// TIA Portal V16 export
// export: Created 2022-11-17T15:49:47.8701163Z, ExportSetting WithDefaults, DisplayName Totally Integrated Automation Portal, DisplayVersion V16 Update 6, DisplayName TIA Portal Version Control Interface, DisplayVersion V16 Update 2, DisplayName TIA Portal Openness, DisplayVersion V16 Update 6, DisplayName SINAMICS Startdrive Advanced, DisplayVersion V16 Update 5, DisplayName SINAMICS Startdrive G130, G150, S120, S150, SINAMICS MV, S210, DisplayVersion V16 Update 5, DisplayName SINAMICS Startdrive G110M, G120, G120C, G120D, G120P, G115D, DisplayVersion V16 Update 5, DisplayName STEP 7 Professional, DisplayVersion V16 Update 6, DisplayName STEP 7 Safety, DisplayVersion V16, DisplayName WinCC Advanced, DisplayVersion V16 Update 6
VAR_GLOBAL   // PLC tag table "Default tag table"
   "E0.4" AT %I0.4 : Bool;   // CONTROLLO SALDATORE FILM
   "E0.5" AT %I0.5 : Bool;   // RICHIESTA APERTURA PORTA
   "E0.6" AT %I0.6 : Bool;   // PRESSOSTATO MACCHINA
   "E0.7" AT %I0.7 : Bool;   // ALLARME TERMICO MACCHINA
   "E1.0" AT %I1.0 : Bool;   // EMERGENZA MACCHINA
   "E1.1" AT %I1.1 : Bool;   // BARRIERE IMPEGNATE ENTRATA
   "E1.2" AT %I1.2 : Bool;   // BARRIERE IMPEGNATE USCITA
   "E1.3" AT %I1.3 : Bool;   // RESET MACCHINA
   "E1.4" AT %I1.4 : Bool;   // MARCIA AUTOMATICA MACCHINA
   "E1.5" AT %I1.5 : Bool;   // ARRESTO MACCHINA
   "E2.0" AT %I2.0 : Bool;   // TAVOLA IN FASE
   "E2.1" AT %I2.1 : Bool;   // [spare] COMANDO FRENO MOTORE ROTAZIONE
   "E2.2" AT %I2.2 : Bool;   // CARRELLO BASSO
   "E2.3" AT %I2.3 : Bool;   // CARRELLO ALTO
   "E2.4" AT %I2.4 : Bool;   // TAGLIO INDIETRO
   "E2.5" AT %I2.5 : Bool;   // TAGLIO AVANTI
   "E2.6" AT %I2.6 : Bool;   // CONTRASTO SALDATORE INDIETRO
   "E2.7" AT %I2.7 : Bool;   // CONTRASTO SALDATORE BASSO
   "E3.0" AT %I3.0 : Bool;   // RISERVA
   "E3.1" AT %I3.1 : Bool;   // RISERVA
   "E3.2" AT %I3.2 : Bool;   // LETTURA CENTRAGGIO PALLET TRASPORTO CENTRO MACCHINA
   "E3.3" AT %I3.3 : Bool;   // CONTEGGIO CENTRAGGIO PALLET TRASPORTO CENTRO MACCHINA
   "E3.4" AT %I3.4 : Bool;   // CONTROLLO ROTAZIONE TAVOLA IN ENTRATA E LETTURA LUNGHEZZA PALLET
   "E3.5" AT %I3.5 : Bool;   // CONTROLLO ROTAZIONE TAVOLA IN USCITA E FINE CICLO
   "E3.6" AT %I3.6 : Bool;   // SEGNALE PALLET PRONTO IN ENTRATA
   "E3.7" AT %I3.7 : Bool;   // SEGNALE PRONTO A RICEVERE IN USCITA
   "E4.0" AT %I4.0 : Bool;   // SEGNALE FINE TRASFERIMENTO PALLET IN USCITA
   "E4.1" AT %I4.1 : Bool;   // SEGNALE ESCLUSIONE FASCIATURA
   "E4.2" AT %I4.2 : Bool;   // POSIZIONAMENTO PALLET TRASPORTO POS. 01
   "E4.3" AT %I4.3 : Bool;   // POSIZIONAMENTO PALLET TRASPORTO POS. 02
   "E4.4" AT %I4.4 : Bool;   // POSIZIONAMENTO PALLET TRASPORTO POS. 03
   "E4.5" AT %I4.5 : Bool;   // POSIZIONAMENTO PALLET TRASPORTO POS. 04
   "E4.6" AT %I4.6 : Bool;   // POSIZIONAMENTO PALLET TRASPORTO POS. 05
   "E5.1" AT %I5.1 : Bool;   // POSIZIONAMENTO PALLET TRASPORTO POS. 08
   "E5.3" AT %I5.3 : Bool;   // [B2783] CONTROLLO 2 POSIZIONAMENTO POS. 05
   "E6.0" AT %I6.0 : Bool;   // CARRELLO BASSO (TOP)
   "E6.1" AT %I6.1 : Bool;   // CARRELLO ALTO (TOP)
   "E6.2" AT %I6.2 : Bool;   // LETTURA ALTEZZA PALLET (TOP)
   "E6.3" AT %I6.3 : Bool;   // PINZA CHIUSA BLOCCO FILM (TOP)
   "E6.4" AT %I6.4 : Bool;   // TAGLIO FILM AVANTI (TOP)
   "E6.5" AT %I6.5 : Bool;   // TAGLIO FILM INDIETRO (TOP)
   "E6.6" AT %I6.6 : Bool;   // ROTTURA ESAURIMENTO FILM (TOP)
   "E7.0" AT %I7.0 : Bool;   // CARRELLO INDIETRO (TOP)
   "E7.1" AT %I7.1 : Bool;   // CARRELLO AVANTI POSIZIONE TAGLIO (TOP)
   "E7.3" AT %I7.3 : Bool;   // PINZA CHIUSA TRAINO FILM (TOP)
   "E7.4" AT %I7.4 : Bool;   // SICUREZZA AVANZAMENTO (TOP)
   "E7.5" AT %I7.5 : Bool;   // SICUREZZA DISCESA (TOP) SX
   "E7.6" AT %I7.6 : Bool;   // SICUREZZA DISCESA (TOP) DX
   "E7.7" AT %I7.7 : Bool;   // SICUREZZA CONTROLLO SGANCIO FRENI SAL.-DISC. (TOP)
   HSC2Value AT %ID1004 : DInt;   // Counter value for HSC2
   HSC1Value AT %ID1000 : DInt;
   "E4.7" AT %I4.7 : Bool;   // POSIZIONAMENTO PALLET TRASPORTO POS. 06
   "E5.0" AT %I5.0 : Bool;   // POSIZIONAMENTO PALLET TRASPORTO POS. 07
   "E5.2" AT %I5.2 : Bool;   // [B2782] CONTROLLO 1 POSIZIONAMENTO POS. 05
   "E5.4" AT %I5.4 : Bool;   // SEGNALE PORTA TAGLIAFUOCO APERTA
   "E5.5" AT %I5.5 : Bool;   // SEGNALE CHIUSURA PORTA TAGLIAFUOCO
   "E5.6" AT %I5.6 : Bool;   // SelectorBypass
   "E5.7" AT %I5.7 : Bool;   // Free
   "E6.7" AT %I6.7 : Bool;   // SPARE - NOT USED
   "E7.2" AT %I7.2 : Bool;   // RISERVA
   "A0.0" AT %Q0.0 : Bool;   // APERTURA PORTA
   "A0.1" AT %Q0.1 : Bool;   // EMERGENZA PLC SU PILZ
   "A0.2" AT %Q0.2 : Bool;   // EMERGENZA MACCHINA
   "A0.3" AT %Q0.3 : Bool;   // MARCIA AUTOMATICA MACCHINA
   "A0.4" AT %Q0.4 : Bool;   // SEGNALATORE ACUSTICO MARCIA
   "A0.6" AT %Q0.6 : Bool;   // FRENO MOTORE ROTAZIONE
   "A0.7" AT %Q0.7 : Bool;   // MOTORE ROTAZIONE
   "A1.0" AT %Q1.0 : Bool;   // FASCIA STRETTA
   "A1.1" AT %Q1.1 : Bool;   // CORDA STRETTA
   "A2.0" AT %Q2.0 : Bool;   // PINZA APERTA
   "A2.1" AT %Q2.1 : Bool;   // PINZA CHIUSA
   "A2.2" AT %Q2.2 : Bool;   // TAGLIO AVANTI / INDIETRO
   "A2.3" AT %Q2.3 : Bool;   // SOFFIO ARIA PER CODA FILM
   "A2.4" AT %Q2.4 : Bool;   // TAGLIO FILM
   "A2.5" AT %Q2.5 : Bool;   // SALDATORE FILM
   "A2.6" AT %Q2.6 : Bool;   // CONTRASTO SALDATORE AVANTI
   "A2.7" AT %Q2.7 : Bool;   // CONTRASTO SALDATORE INDIETRO
   "A3.0" AT %Q3.0 : Bool;   // CONTRASTO SALDATORE SALITA/DISCESA
   "A3.1" AT %Q3.1 : Bool;   // RISERVA
   "A3.2" AT %Q3.2 : Bool;   // RISERVA
   "A3.3" AT %Q3.3 : Bool;   // MOTORE TRASPORTO CENTRO MACCHINA
   "A3.4" AT %Q3.4 : Bool;   // SEGNALE PRONTO A RICEVERE IN ENTRATA
   "A3.5" AT %Q3.5 : Bool;   // SEGNALE FINE TRASFERIMENTO PALLET IN ENTRATA
   "A3.6" AT %Q3.6 : Bool;   // SEGNALE PALLET PRONTO IN USCITA
   "A3.7" AT %Q3.7 : Bool;   // SEGNALE PRONTO PER CHIUSURA PORTA TAGLIAFUOCO
   "A4.0" AT %Q4.0 : Bool;   // MOTORE TRASPORTO POS. 01 AVANTI
   "A4.1" AT %Q4.1 : Bool;   // MOTORE TRASPORTO POS. 02 AVANTI
   "A4.2" AT %Q4.2 : Bool;   // MOTORE TRASPORTO POS. 03 AVANTI
   "A4.3" AT %Q4.3 : Bool;   // MOTORE TRASPORTO POS. 04 AVANTI
   "A4.4" AT %Q4.4 : Bool;   // MOTORE TRASPORTO POS. 05 AVANTI
   "A4.5" AT %Q4.5 : Bool;   // MOTORE TRASPORTO POS. 06 AVANTI
   "A4.6" AT %Q4.6 : Bool;   // MOTORE TRASPORTO POS. 07 AVANTI
   "A4.7" AT %Q4.7 : Bool;   // MOTORE TRASPORTO POS. 08 AVANTI
   "A5.0" AT %Q5.0 : Bool;   // Lamp By-pass
   "A5.1" AT %Q5.1 : Bool;   // SPARE - NOT USED
   "A5.2" AT %Q5.2 : Bool;   // SPARE - NOT USED
   "A5.3" AT %Q5.3 : Bool;   // SPARE - NOT USED
   "A6.0" AT %Q6.0 : Bool;   // MOTORE CARRELLO (TOP) AVANTI
   "A6.1" AT %Q6.1 : Bool;   // MOTORE CARRELLO (TOP) INDIETRO
   "A6.2" AT %Q6.2 : Bool;   // START INVERTER SALITA CARRELLO (TOP)
   "A6.3" AT %Q6.3 : Bool;   // START INVERTER DISCESA CARRELLO (TOP)
   "A6.4" AT %Q6.4 : Bool;   // FRENO MOTORE (TOP) SALITA/DISCESA
   "A6.5" AT %Q6.5 : Bool;   // PINZA APERTA BLOCCO FILM (TOP)
   "A6.6" AT %Q6.6 : Bool;   // PINZA CHIUSA BLOCCO FILM (TOP)
   "A6.7" AT %Q6.7 : Bool;   // TAGLIO FILM AVANTI (TOP)
   "A7.0" AT %Q7.0 : Bool;   // TAGLIO FILM INDIETRO (TOP)
   "A7.1" AT %Q7.1 : Bool;   // PINZA APERTA TRAINO FILM (TOP)
   "A7.2" AT %Q7.2 : Bool;   // PINZA CHIUSA TRAINO FILM (TOP)
   "A5.4" AT %Q5.4 : Bool;   // SPARE - NOT USED
   "A5.5" AT %Q5.5 : Bool;   // SPARE - NOT USED
   "A5.6" AT %Q5.6 : Bool;   // SPARE - NOT USED
   "A0.5" AT %Q0.5 : Bool;   // ENABLE INVERTER ROTAZIONE
   "A5.7" AT %Q5.7 : Bool;   // SPARE - NOT USED
   "A10.0" AT %Q10.0 : Bool;   // SPARE - NOT USED
   "A10.1" AT %Q10.1 : Bool;   // SPARE - NOT USED
   "A10.2" AT %Q10.2 : Bool;   // SPARE - NOT USED
   "A10.3" AT %Q10.3 : Bool;   // SPARE - NOT USED
   "A7.3" AT %Q7.3 : Bool;   // SPARE - NOT USED
   "A7.4" AT %Q7.4 : Bool;   // SPARE - NOT USED
   "A7.5" AT %Q7.5 : Bool;   // SPARE - NOT USED
   "A7.6" AT %Q7.6 : Bool;   // SPARE - NOT USED
   "A7.7" AT %Q7.7 : Bool;   // SPARE - NOT USED
   "M0.0" AT %M0.0 : Bool;   // Machine cycle: M0.0 Start cycle
   "M0.1" AT %M0.1 : Bool;   // Machine cycle: M0.1 Waiting for top before
   "M0.2" AT %M0.2 : Bool;   // Machine cycle: M0.2 Loading data for spool carriage position
   "M0.3" AT %M0.3 : Bool;   // Machine cycle: M0.3 Waiting for pressure plate and lifter
   "M0.4" AT %M0.4 : Bool;   // Machine cycle: M0.4 Spool carriage upward/downward with rotation
   "M0.5" AT %M0.5 : Bool;   // Machine cycle: M0.5 Table rotation - Table revolution counter
   "M0.6" AT %M0.6 : Bool;   // Machine cycle: M0.6 Load new data for next spool carriage height
   "M0.7" AT %M0.7 : Bool;   // Machine cycle: M0.7 Spool carriage upward/downward with rotation
   "M1.0" AT %M1.0 : Bool;   // Machine cycle: M1.0 Revolution over welder contrast
   "M1.1" AT %M1.1 : Bool;   // Machine cycle: M1.1
   "M1.2" AT %M1.2 : Bool;   // Machine cycle: M1.2 Table rotation deceleration
   "M1.3" AT %M1.3 : Bool;   // Machine cycle: M1.3 Table rotation deceleration
   "M1.4" AT %M1.4 : Bool;   // Machine cycle: M1.4 Stop table rotation - Waiting step
   "M1.5" AT %M1.5 : Bool;   // Machine cycle: M1.5 Waiting step
   "M1.6" AT %M1.6 : Bool;   // Machine cycle: M1.6 Pallet unload
   "M1.7" AT %M1.7 : Bool;   // Machine cycle: M1.7 Clamp and top check
   "M2.0" AT %M2.0 : Bool;   // Machine cycle: V2.0 Label cycle 1st label
   "M2.2" AT %M2.2 : Bool;   // Machine cycle: M2.2 Clamp and top check (Test cycle)
   "M2.3" AT %M2.3 : Bool;   // Machine cycle: M2.3 Checking step (Test cycle)
   "M2.4" AT %M2.4 : Bool;   // Label cycle
   "M3.0" AT %M3.0 : Bool;   // Machine cycle: M3.0 Table rotation middle speed
   "M3.1" AT %M3.1 : Bool;   // Machine cycle: M3.1 Table rotation deceleration
   "M3.2" AT %M3.2 : Bool;   // Machine cycle: M3.2 Table rotation deceleration
   "M3.3" AT %M3.3 : Bool;   // Machine cycle: M3.3 Waiting for top cycle
   "M5.0" AT %M5.0 : Bool;   // Top cycle: V5.0 Start cycle
   "M5.1" AT %M5.1 : Bool;   // Top cycle: V5.1 Closing clamp to pull top film
   "M5.2" AT %M5.2 : Bool;   // Top cycle: V5.2 Opening clamp to block top film
   "M5.3" AT %M5.3 : Bool;   // Top cycle: V5.3 Top carriage forward
   "M5.4" AT %M5.4 : Bool;   // Top cycle: V5.4 Closing clamp to block top film
   "M5.5" AT %M5.5 : Bool;   // Top cycle: V5.5 Top carriage down
   "M5.6" AT %M5.6 : Bool;   // Top cycle: V5.6 Top carriage on pallet top
   "M5.7" AT %M5.7 : Bool;   // Top cycle: V5.7 Top cutter forward
   "M6.0" AT %M6.0 : Bool;   // Top cycle: V6.0 Top cutter backward
   "M6.1" AT %M6.1 : Bool;   // Top cycle: V6.1 Top carriage forward\Top cutter backward
   "M6.2" AT %M6.2 : Bool;   // Top cycle: V6.2 Top carriage downward to pull down top film
   "M6.3" AT %M6.3 : Bool;   // Top cycle: V6.3 Top carriage downward to release top film
   "M6.4" AT %M6.4 : Bool;   // Top cycle: V6.4 Top carriage stopped against vibration
   "M6.5" AT %M6.5 : Bool;   // Top cycle: V6.5 Top carriage upward
   "M6.6" AT %M6.6 : Bool;   // Top cycle: V6.6 Top carriage upward and backward
   "M6.7" AT %M6.7 : Bool;   // Top cycle: V6.7 Waiting for Rotoplat end cycle
   "M8.0" AT %M8.0 : Bool;   // Top film ended cycle: V8.0 Top carriage backward
   "M8.1" AT %M8.1 : Bool;   // Top film ended cycle: V8.1 Top carriage downward
   "M8.2" AT %M8.2 : Bool;   // Top film ended cycle: V8.2 Top carriage forward
   "M8.3" AT %M8.3 : Bool;   // Top film ended cycle: V8.3 Wait for reset button
   "M8.4" AT %M8.4 : Bool;   // Top film ended cycle: V8.4 Wait for automatic mode
   "M8.5" AT %M8.5 : Bool;   // Top film ended cycle: V8.5 Top carriage backward
   "M8.6" AT %M8.6 : Bool;   // Top film ended cycle: V8.6 Top carriage upward
   "M9.0" AT %M9.0 : Bool;   // Top cycle: V9.0 Top carriage downward for 90 degree top
   "M9.1" AT %M9.1 : Bool;   // Top cycle: V9.1 Wait step 1 for 90 degree top
   "M9.2" AT %M9.2 : Bool;   // Top cycle: V9.2 Top carriage upward for 90 degree top
   "M9.3" AT %M9.3 : Bool;   // Top cycle: V9.3 Wait step 2 for 90 degree top
   "M9.4" AT %M9.4 : Bool;   // Top cycle: V9.4 Waiting step 3 for 90 degree top after top
   "M9.5" AT %M9.5 : Bool;   // Top cycle: V9.5 Top carriage upward for 90 degree top
   "M9.6" AT %M9.6 : Bool;   // Top cycle: V9.6 Wait step 4 for 90 degree top after top
   Alarm AT %M10.0 : Bool;   // Main emergency
   "M10.1" AT %M10.1 : Bool;   // Prearrangement automatic cycle
   Manu AT %M10.2 : Bool;   // Manual mode
   Auto AT %M10.3 : Bool;   // Automatic mode
   "M10.4" AT %M10.4 : Bool;   // Automatic mode for film ended or broken
   Stop AT %M10.5 : Bool;   // Memory stop cycle
   "M10.6" AT %M10.6 : Bool;   // Memory to stop cycle for door open request
   Warning AT %M10.7 : Bool;   // Warning message active
   "M11.5" AT %M11.5 : Bool;   // Button Reset support memory
   "M11.6" AT %M11.6 : Bool;   // Memory release Button Reset
   FilmEnd AT %M12.0 : Bool;   // Film ended or broken
   TopEnd AT %M12.1 : Bool;   // Top film ended or broken
   On AT %M12.7 : Bool;   // Bit always on
   "M14.7" AT %M14.7 : Bool;   // Table rotation backward to reset encoder
   Reset AT %M15.0 : Bool;   // Main reset
   "M15.1" AT %M15.1 : Bool;   // Request to reset spool carriage encoder
   "M15.2" AT %M15.2 : Bool;   // First cycle
   TransitIn AT %M15.3 : Bool;   // Pallet transit in infeed
   TransitOut AT %M15.4 : Bool;   // Pallet transit in outfeed
   TransitInBkw AT %M15.5 : Bool;   // Transit memory in infeed from reverse
   V15_6 AT %M15.6 : Bool;   // Automatic mode for external conveyors
   "M15.7" AT %M15.7 : Bool;   // Request to reset table rotation encoder
   "M16.0" AT %M16.0 : Bool;   // Conveyor cycle: M16.0 Start cycle
   "M16.1" AT %M16.1 : Bool;   // Conveyor cycle: M16.1 Loading pallet
   "M16.2" AT %M16.2 : Bool;   // Conveyor cycle: M16.2 Pallet positioned
   "M16.3" AT %M16.3 : Bool;   // Conveyor cycle: M16.3 Unloading pallet
   "M16.4" AT %M16.4 : Bool;   // Conveyor cycle: M16.4 Loading/unloading pallet simultaneously
   "M16.5" AT %M16.5 : Bool;   // Conveyor cycle: M16.5 Unloading pallet
   "M16.6" AT %M16.6 : Bool;   // Conveyor cycle: M16.6 Loading pallet from reverse
   "M16.7" AT %M16.7 : Bool;   // Conveyor cycle: M16.7 Pallet positioned from reverse
   "M17.0" AT %M17.0 : Bool;   // Pallet load cycle: V17.0 Table rotation to load phase
   "M17.1" AT %M17.1 : Bool;   // Pallet load cycle: V17.1 Table rotation to machine phase from load
   "M17.2" AT %M17.2 : Bool;   // Pallet load cycle: V17.2 Table rotation to unload phase
   "M17.3" AT %M17.3 : Bool;   // Pallet load cycle: V17.3 Table rotation to machine phase from unload
   "M17.4" AT %M17.4 : Bool;   // Pallet load cycle: V17.4 Table rotation to reverse phase
   "M17.5" AT %M17.5 : Bool;   // Pallet load cycle: V17.5 Table rotation to machine phase from re
   "M18.0" AT %M18.0 : Bool;   // Ring clamp cycle: M18.0 Start cycle
   "M18.1" AT %M18.1 : Bool;   // Ring clamp cycle: M18.1 Open clamp
   "M18.2" AT %M18.2 : Bool;   // Ring clamp cycle: M18.2 Waiting for welder contrast up
   "M18.3" AT %M18.3 : Bool;   // Ring clamp cycle: M18.3 Waiting table deceleration
   "M18.4" AT %M18.4 : Bool;   // Ring clamp cycle: M18.4 Ring clamp upward
   "M18.5" AT %M18.5 : Bool;   // Ring clamp cycle: M18.5 Opening ring clamp
   "M18.6" AT %M18.6 : Bool;   // Ring clamp cycle: M18.6 Waiting for table rotation in phase
   "M18.7" AT %M18.7 : Bool;   // Ring clamp cycle: M18.7 Closing ring clamp
   "M19.0" AT %M19.0 : Bool;   // Ring clamp cycle: M19.0 Welder and cut unit upward
   "M19.1" AT %M19.1 : Bool;   // Ring clamp cycle: M19.1 Waiting for welding time
   "M19.2" AT %M19.2 : Bool;   // Ring clamp cycle: M19.2 Welder unit downward
   "M19.3" AT %M19.3 : Bool;   // Ring clamp cycle: M19.3 Waiting for pallet unload
   "M20.0" AT %M20.0 : Bool;   // Claw clamp HS40 cycle: M20.0 Start cycle
   "M20.1" AT %M20.1 : Bool;   // Claw clamp HS40 cycle: M20.1 Opening clamp
   "M20.2" AT %M20.2 : Bool;   // Claw clamp HS40 cycle: M20.2 Waiting for table rotation in phase
   "M20.3" AT %M20.3 : Bool;   // Claw clamp HS40 cycle: M20.3 Closing clamp
   "M20.4" AT %M20.4 : Bool;   // Claw clamp HS40 cycle: M20.4 Welder and cut unit forward
   "M20.5" AT %M20.5 : Bool;   // Claw clamp HS40 cycle: M20.5 Waiting for cut and welding time
   "M20.6" AT %M20.6 : Bool;   // Claw clamp HS40 cycle: M20.6 Welder and cut unit backward
   "M22.0" AT %M22.0 : Bool;   // Spring clamp cycle: M22.0 Start cycle
   "M22.1" AT %M22.1 : Bool;   // Spring clamp cycle: M22.1 Open clamp
   "M22.2" AT %M22.2 : Bool;   // Spring clamp cycle: M22.2 Waiting for welder contrast up
   "M22.3" AT %M22.3 : Bool;   // Spring clamp cycle: M22.3 Waiting table deceleration
   "M22.4" AT %M22.4 : Bool;   // Spring clamp cycle: M22.4 Spring clamp upward
   "M22.5" AT %M22.5 : Bool;   // Spring clamp cycle: M22.5 Opening spring clamp
   "M22.6" AT %M22.6 : Bool;   // Spring clamp cycle: M22.6 Waiting for table rotation in phase
   "M22.7" AT %M22.7 : Bool;   // Spring clamp cycle: M22.7 Table rotation forward for twist
   "M23.0" AT %M23.0 : Bool;   // Spring clamp cycle: M23.0 Closing spring clamp
   "M23.1" AT %M23.1 : Bool;   // Spring clamp cycle: M23.1 Welder and cut unit upward
   "M23.2" AT %M23.2 : Bool;   // Spring clamp cycle: M23.2 Waiting for welding time
   "M23.3" AT %M23.3 : Bool;   // Spring clamp cycle: M23.3 Welder unit downward
   "M23.4" AT %M23.4 : Bool;   // Spring clamp cycle: M23.4 Waiting for welder contrast down
   "M30.0" AT %M30.0 : Bool;   // Film broken cycle: M30.0 Start cycle
   "M30.1" AT %M30.1 : Bool;   // Film broken cycle: M30.1 All unit to home position
   "M30.2" AT %M30.2 : Bool;   // Film broken cycle: M30.2 Spool carriage to film change position
   "M30.3" AT %M30.3 : Bool;   // Film broken cycle: M30.3 Waiting for alarm mode
   "M30.4" AT %M30.4 : Bool;   // Film broken cycle: M30.4 Waiting automatic mode
   "M30.5" AT %M30.5 : Bool;   // Film broken cycle: M30.5 Spool carriage downward
   "M30.6" AT %M30.6 : Bool;   // Film broken cycle: M30.6 Waiting step
   "M32.0" AT %M32.0 : Bool;   // Film broken cycle 1: M32.0 Start cycle
   "M32.1" AT %M32.1 : Bool;   // Film broken cycle 1: M32.1 Table rotation middle speed
   "M32.2" AT %M32.2 : Bool;   // Film broken cycle 1: M32.2 Table rotation middle speed
   "M32.3" AT %M32.3 : Bool;   // Film broken cycle 1: M32.3 Table rotation deceleration
   "M32.4" AT %M32.4 : Bool;   // Film broken cycle 1: M32.4 Table rotation deceleration
   "M32.5" AT %M32.5 : Bool;   // Film broken cycle 1: M32.5 Waiting step
   V50_1 AT %M50.1 : Bool;   // Infeed conveyor pos.1 load
   V50_6 AT %M50.6 : Bool;   // Transit memory pos6->pos7
   V51_1 AT %M51.1 : Bool;   // Memory to exclude wrapping in pos 1
   V56_0 AT %M56.0 : Bool;   // Start cycle lifter pos.2: V56.0 Lifter empty and low
   V56_1 AT %M56.1 : Bool;   // Start cycle lifter pos.2: V56.1 Lifter upstroke
   V56_2 AT %M56.2 : Bool;   // Start cycle lifter pos.2: V56.2 Waiting step - pallet load
   V56_3 AT %M56.3 : Bool;   // Start cycle lifter pos.2: V56.3 Lifter downstroke
   V56_4 AT %M56.4 : Bool;   // Start cycle lifter pos.2: V56.4 Waiting step - pallet unload
   V56_5 AT %M56.5 : Bool;   // Start cycle lifter pos.2: V56.5
   V56_6 AT %M56.6 : Bool;   // Start cycle lifter pos.2: V56.6
   V57_0 AT %M57.0 : Bool;   // Load to pos1 with forklift request
   V57_1 AT %M57.1 : Bool;   // Load to pos1 with forklift ok
   V57_2 AT %M57.2 : Bool;   // Unload from pos1 with forklift request
   V57_3 AT %M57.3 : Bool;   // Unload from pos1 with forklift OK
   V57_5 AT %M57.5 : Bool;   // Start cycle pos.1 OK
   Sgn_TopPosizTransfer AT %M64.1 : Bool;   // Top Out Supp. Out - Signal " Top In Position for Pallet Transfe
   ContrastCarriageOk1 AT %M70.0 : Bool;   // ContrastCarriageOK1: Contrast carriage in position to return to start cycle
   ContrastCarriageOk4 AT %M70.3 : Bool;   // ContrastCarriageOk4: Contrast carriage in position for film broken cycle
   ContrastCarriageOk7 AT %M70.6 : Bool;   // ContrastCarriageOk7: Contrast carriage unit in position to begin cycle
   ContrastCarriageOk17 AT %M72.0 : Bool;   // ContrastCarriageOk17: Contrast carriage in position for pallet transit
   ClampCutOk1 AT %M80.0 : Bool;   // ClampCutOK1: Clamp and cutter in position to return to start cycle
   ClampCutOk2 AT %M80.1 : Bool;   // ClampCutOK2: Film tail wrapped
   ClampCutOk3 AT %M80.2 : Bool;   // ClampCutOK3: Main emergency (1+) for welder circuit control
   ClampCutOk4 AT %M80.3 : Bool;   // ClampCutOk4: Clamp in position for film broken cycle
   ClampCutOk5 AT %M80.4 : Bool;   // ClampCutOk5: Revolution over welder contrast done
   ClampCutOk6 AT %M80.5 : Bool;   // ClampCutOk6: Clamp and cutter cycle ended
   ClampCutOk7 AT %M80.6 : Bool;   // ClampCutOk7: Clamp and cutter units in position to begin cycle
   ClampCutOk8 AT %M80.7 : Bool;   // ClampCutOk8: Table rotation middle speed
   ClampCutOk9 AT %M81.0 : Bool;
   ClampCutOk10 AT %M81.1 : Bool;   // ClampCutOk10: Clamp and cut unit in safety position for table rotation
   ClampCutOK11 AT %M81.2 : Bool;   // ClampCutOk11: Exclude deceleration not correct alarm
   ClampCutOK12 AT %M81.3 : Bool;   // ClampCutOk12: Film request during clamp cycle
   ClampCutOk13 AT %M81.4 : Bool;   // ClampCutOk13: Request to move spool carrage up at the begining
   ClampCutOk14 AT %M81.5 : Bool;   // ClampCutOk14: Ok to move spool carrage down at the begining
   ClampCutOk15 AT %M81.6 : Bool;   // ClampCutOk15: Request to move spool carrage up to cover film tail
   ClampCutOk16 AT %M81.7 : Bool;   // ClampCutOk16: Ok to move spool carrage down to cover film tail
   ClampCutOk17 AT %M82.0 : Bool;   // ClampCutOk17: Clamp units in position for pallet transit
   ClampCutOk18 AT %M82.1 : Bool;   // ClampCutOk18: Enable for spool carriage downward at cycle end
   ClampCutOk19 AT %M82.2 : Bool;   // ClampCutOk19: Clamp and cut unit in safety position for pallet lifter
   ClampCutOk20 AT %M82.3 : Bool;   // Pallet backward request for ClampCut cycle
   ClampCutOk21 AT %M82.4 : Bool;   // ClampCutOk21: Cutter arm forward
   "M83.0" AT %M83.0 : Bool;   // Table rotation forward for twist
   "M83.1" AT %M83.1 : Bool;   // Table rotation backward for twist
   LifterOK1 AT %M84.0 : Bool;   // LifterOK1: Pallet lifter down
   LifterOk2 AT %M84.1 : Bool;   // LifterOk2: Pallet lifter up
   "M84.3" AT %M84.3 : Bool;   // Pallet lifter upward
   "M84.4" AT %M84.4 : Bool;   // Pallet lifter downward
   RopeUnitOk1 AT %M84.5 : Bool;   // RopeUnitOk1: Rope unit open
   RopeUnitOk2 AT %M84.6 : Bool;   // RopeUnitOk2: Full rope unit open
   TopOK1 AT %M85.0 : Bool;   // Top carriage OK1: Top cycle ended
   TopOK2 AT %M85.1 : Bool;   // Top carriage OK2: Ok for pressure plate downward on 90 degree top
   TopOK3 AT %M85.2 : Bool;   // Top carriage OK3: Top carriage backward or forward
   TopOk4 AT %M85.3 : Bool;   // Top carriage OK4: Top carriage up
   TopOk5 AT %M85.6 : Bool;   // Top carriage OK5: Top cycle ended for top dustproof
   TopOk6 AT %M85.7 : Bool;   // Top carriage OK6: Emergency rele' on pilz chain
   PressureOk1 AT %M86.0 : Bool;   // PressureOk1: Pressure plate on pallet
   PressureOk2 AT %M86.1 : Bool;   // PressureOk2: Pressure plate up
   PressureOk3 AT %M86.2 : Bool;   // PressureOk3: Pressure plate Ok for pallet height
   "M86.3" AT %M86.3 : Bool;   // Pressure plate downward
   "M86.4" AT %M86.4 : Bool;   // Pressure plate upward
   V86_5 AT %M86.5 : Bool;   // Pressure Plate downstroke request
   V87_0 AT %M87.0 : Bool;   // Top carriage forward
   V87_1 AT %M87.1 : Bool;   // Top carriage backward
   V87_2 AT %M87.2 : Bool;   // Top carriage forward/backward slow speed
   V87_3 AT %M87.3 : Bool;   // Table rotation forward for top
   V87_4 AT %M87.4 : Bool;   // Table rotation backward for top
   TopOk7 AT %M88.0 : Bool;   // TopOk7: Top carriage backward
   TopOk8 AT %M88.1 : Bool;   // TopOK8: All top units in position for automatic cycle
   TopOk9 AT %M88.2 : Bool;   // TopOk3: Top before cycle ended
   TopOk10 AT %M88.4 : Bool;   // TopOk10: Table rotation middle speed
   TopOk11 AT %M88.5 : Bool;   // Top carriage OK11: All top units OK for automatic cycle
   TopOk12 AT %M88.6 : Bool;   // Top carriage OK12: Carriage downward for top 90 ended cycle
   V89_0 AT %M89.0 : Bool;   // Table rotation for top cycle (Top->Table)
   V89_1 AT %M89.1 : Bool;   // Fast speed table rotation for top cycle (Top->Table)
   V89_2 AT %M89.2 : Bool;   // Middle speed table rotation for top cycle (Top->Table)
   V89_3 AT %M89.3 : Bool;   // Spool carriage downward for top cycle (Top->Table)
   V89_4 AT %M89.4 : Bool;   // Spool carriage upward for top cycle (Top->Table)
   V89_5 AT %M89.5 : Bool;   // Memory to control the top cycle reset (Top->Table)
   Top_OFF AT %M89.6 : Bool;   // Top off by the machine configuration
   Top_ON AT %M89.7 : Bool;   // Top on by the machine configuration
   ConvOk1 AT %M90.0 : Bool;   // ConvOk1: Pallet ready to be wrapped
   ConvOk2 AT %M90.1 : Bool;   // ConvOk2: Pallet in position to return to start cycle
   ConvOk3 AT %M90.2 : Bool;   // ConvOk3: Conveyor is running
   ConvOk4 AT %M90.3 : Bool;   // ConvOk4: Forward for inverter
   ConvOk5 AT %M90.4 : Bool;   // ConvOK5: Fast speed for conveyor
   ConvOk6 AT %M90.5 : Bool;   // ConvOk6: Slow speed for conveyor
   ConvOk7 AT %M90.6 : Bool;   // ConvOk7: Backward for inverter
   V90_7 AT %M90.7 : Bool;   // ConvOk8: Conveyor is running
   "M91.0" AT %M91.0 : Bool;   // Load data from table to display
   "M91.1" AT %M91.1 : Bool;   // Load data from display to table
   "M91.2" AT %M91.2 : Bool;   // Program active is Ok
   TechnoplatOk1 AT %M92.0 : Bool;   // TechnoplatOk1: All unit to home position
   TechnoplatOk2 AT %M92.1 : Bool;   // TechnoplatOk2: Reset all cycle
   TechnoplatOk3 AT %M92.2 : Bool;   // TechnoplatOk3: A manual operation has been done
   TechnoplatOk4 AT %M92.3 : Bool;   // TechnoplatOk4: Top unit is able to start his cycle
   TechnoplatOk5 AT %M92.4 : Bool;   // TechnoplatOk5:
   TechnoplatOk6 AT %M92.5 : Bool;   // TechnoplatOk6:
   "M93.0" AT %M93.0 : Bool;   // One shot rising (OSR) for table phase sensor
   "M93.1" AT %M93.1 : Bool;   // One shot falliing (OSF) for table phase sensor
   StopRequest AT %M93.5 : Bool;   // (Memory) Stop request by operator button
   V94_0 AT %M94.0 : Bool;   // Spool carriage upward request for table cycle
   V94_1 AT %M94.1 : Bool;   // Spool carriage downward request for table cycle
   E01 AT %M100.0 : Bool;   // Spool carriage encoder channel A (Technoplat)
   E02 AT %M100.1 : Bool;   // Spool carriage encoder channel B (Technoplat)
   E03_NotUsed AT %M100.2 : Bool;   // Safety barriers excluded by selector (Barrier)
   E04 AT %M100.3 : Bool;   // Infeed safety barrier engaged (Barrier)
   E05 AT %M100.4 : Bool;   // Outfeed safety barrier engaged (Barrier)
   E06 AT %M100.5 : Bool;   // Reset button (Technoplat)
   E07_NotUsed AT %M100.6 : Bool;   // Key selector automatic (0)/manual (1) mode (Technoplat)
   E08 AT %M100.7 : Bool;   // Automatic functioning button (Technoplat)
   E09 AT %M101.0 : Bool;   // Stop request by operator button (Technoplat)
   E10 AT %M101.1 : Bool;   // Request to open door key selector (1 open) (Technoplat)
   E11 AT %M101.2 : Bool;   // Pressure switch (Technoplat)
   E12 AT %M101.3 : Bool;   // Thermic alarm (Technoplat)
   E13 AT %M101.4 : Bool;   // Fault inverter (Technoplat)
   E14 AT %M101.5 : Bool;   // Emergency stop push button (Technoplat)
   E15 AT %M101.6 : Bool;   // Main emergency 1+ (Technoplat)
   E16 AT %M101.7 : Bool;   // Spool carriage down (Technoplat)
   E17 AT %M102.0 : Bool;   // Spool carriage up (Technoplat)
   E18 AT %M102.1 : Bool;   // Reading pallet height on spool carriage (Technoplat)
   E19 AT %M102.2 : Bool;   // Film broken or ended on spool carriage (Technoplat)
   E20 AT %M102.3 : Bool;   // Film at 10% on spool carriage (Technoplat)
   E21_NotUsed AT %M102.4 : Bool;   // Reading pallet height on spool carriage with reflector (Technoplat)
   E22 AT %M102.5 : Bool;   // Table rotation phase sensor (Technoplat)
   E23_NotUsed AT %M102.6 : Bool;   // Pallet lifter down (Lifter)
   E24 AT %M102.7 : Bool;   // Pressure plate up (Pressure plate)
   E25 AT %M103.0 : Bool;   // Single rope unit open (Rope unit)
   E26_NotUsed AT %M103.1 : Bool;   // Table rotation phase 2 sensor for top (Technoplat)
   E27_NotUsed AT %M103.2 : Bool;   // Upper(double) rope unit open (Rope unit)
   E28 AT %M103.3 : Bool;   // Pressure plate positioning
   E29 AT %M103.4 : Bool;   // Table rotation load phase sensor (Technoplat)
   E30 AT %M103.5 : Bool;   // Table rotation unload phase sensor (Technoplat)
   E31 AT %M103.6 : Bool;   // Lower (double) rope unit closed (Rope unit)
   E32 AT %M103.7 : Bool;
   E33 AT %M104.0 : Bool;   // Scanner start pushbutton (pos2)
   E34 AT %M104.1 : Bool;   // Labeler start pushbutton (pos3)
   E35 AT %M104.2 : Bool;   // SelectotBypass
   E36 AT %M104.3 : Bool;
   E37 AT %M104.4 : Bool;   // Infeed table rotation control (Conveyor)
   E38 AT %M104.5 : Bool;   // Pallet position control in infeed (Conveyor)
   E39 AT %M104.6 : Bool;   // Pallet position control in outfeed (Conveyor)
   E40 AT %M104.7 : Bool;   // Outfeed table rotation control-End of cycle (Conveyor)
   E41 AT %M105.0 : Bool;   // Pallet position forward (Conveyor)
   E42 AT %M105.1 : Bool;
   E43 AT %M105.2 : Bool;   // Pallet ready in infeed signal (Std signal)
   E44 AT %M105.3 : Bool;   // Ready to receive pallet from outfeed signal (Std signal)
   E45 AT %M105.4 : Bool;   // End of pallet transfer signal (Std signal)
   E46 AT %M105.5 : Bool;   // Wrapping excluded signal (Std signal)
   E47 AT %M105.6 : Bool;   // Pallet ready from reverse
   E48 AT %M105.7 : Bool;
   E49 AT %M106.0 : Bool;   // Wrapping excluded signal (Std signal)
   E50 AT %M106.1 : Bool;
   E51 AT %M106.2 : Bool;   // Signal 1 for program selection by external signal (Std Signal)
   E52 AT %M106.3 : Bool;   // Signal 2 for program selection by external signal (Std Signal)
   E53 AT %M106.4 : Bool;   // Signal 3 for program selection by external signal (Std Signal)
   E54 AT %M106.5 : Bool;   // Signal 4 for program selection by external signal (Std Signal)
   E55_NotUsed AT %M106.6 : Bool;   // Customer conveyor stopped signal (No conveyor signal)
   E56_NotUsed AT %M106.7 : Bool;   // Start wrapping signal (No conveyor signal)
   E57 AT %M107.0 : Bool;
   E58 AT %M107.1 : Bool;
   E59 AT %M107.2 : Bool;   // Coil for welder control (All clamp)
   E60 AT %M107.3 : Bool;   // Film clamp closed (RingSpring clamp)
   E61 AT %M107.4 : Bool;   // Film clamp open (Ring clamp)
   E62_NotUsed AT %M107.5 : Bool;   // Film clamp down (RingSpring clamp)
   E63_NotUsed AT %M107.6 : Bool;   // Film clamp up (Ring clamp)
   E64 AT %M107.7 : Bool;   // Welder contrast down (RingSpring clamp)
   E65 AT %M108.0 : Bool;   // Welder contrast back (Contrast carriage)
   E66 AT %M108.1 : Bool;   // Welder unit down (RingSpring clamp)
   E67 AT %M108.2 : Bool;   // Welder unit up (Ring clamp)
   E68 AT %M108.3 : Bool;   // Clamp carriage forward (Spring clamp)
   E69 AT %M108.4 : Bool;   // Clamp carriage backward (Spring clamp)
   E70 AT %M108.5 : Bool;   // Clamp carriage positioning (Spring clamp)
   E71 AT %M108.6 : Bool;   // Cutting and welding unit forward (Claw clamp)
   E72 AT %M108.7 : Bool;   // Cutting and welding unit backward (Claw clamp)
   E73 AT %M109.0 : Bool;   // Welder unit backward (Claw clamp)
   E74 AT %M109.1 : Bool;
   E75 AT %M109.2 : Bool;
   E76 AT %M109.3 : Bool;
   E77 AT %M109.4 : Bool;
   E78 AT %M109.5 : Bool;
   E79 AT %M109.6 : Bool;
   E80 AT %M109.7 : Bool;
   E81_NotUsed AT %M110.0 : Bool;   // Encoder (Robopac gear) for selfcenter system on preload sysyem (Conveyor)
   E82 AT %M110.1 : Bool;   // Encoder (Robopac gear) for selfcenter system (Conveyor)
   E83 AT %M110.2 : Bool;   // Deceleration for pallet position (Conveyor)
   E84 AT %M110.3 : Bool;   // Pallet positioning for selfcenter system (Conveyor)
   E85 AT %M110.4 : Bool;
   E86 AT %M110.5 : Bool;   // Infeed safety barrier photocell for muting by plc (Barrier)
   E87 AT %M110.6 : Bool;   // Outfeed safety barrier photocell for muting by plc (Barrier)
   E88 AT %M110.7 : Bool;
   E89 AT %M111.0 : Bool;
   E90 AT %M111.1 : Bool;
   E91 AT %M111.2 : Bool;
   E92 AT %M111.3 : Bool;
   E93 AT %M111.4 : Bool;
   E94 AT %M111.5 : Bool;
   E95 AT %M111.6 : Bool;
   E96 AT %M111.7 : Bool;
   E97 AT %M112.0 : Bool;   // Top carriage up (Top)
   E98 AT %M112.1 : Bool;   // Top carriage down (Top)
   E99 AT %M112.2 : Bool;   // Top carriage backward (Top)
   E100 AT %M112.3 : Bool;   // Top carriage forward (Top)
   E101 AT %M112.4 : Bool;   // Reading pallet height for top carriage (Top)
   E102 AT %M112.5 : Bool;   // Safety for top carriage movement (Top)
   E103 AT %M112.6 : Bool;   // Top film cutter forward (Top)
   E104 AT %M112.7 : Bool;   // Top film cutter backward (Top)
   E105 AT %M113.0 : Bool;   // Clamp to block top film closed (Top)
   E106 AT %M113.1 : Bool;   // Clamp to pull top film closed (Top)
   E107 AT %M113.2 : Bool;   // Top film ended sensor (Top)
   E108 AT %M113.3 : Bool;   // Safety for top carriage downward for infeed conveyor (Top)
   E109 AT %M113.4 : Bool;   // Safety for top carriage downward for outfeed conveyor (Top)
   E110 AT %M113.5 : Bool;   // Top carriage position under pressure plate (Top)
   E111 AT %M113.6 : Bool;   // Top carriage brake control (1 braked) (Top)
   E112 AT %M113.7 : Bool;
   E113 AT %M114.0 : Bool;
   E114 AT %M114.1 : Bool;
   E115 AT %M114.2 : Bool;
   E116 AT %M114.3 : Bool;
   E117 AT %M114.4 : Bool;   // SEGNALE PORTA TAGLIAFUOCO APERTA
   E118 AT %M114.5 : Bool;   // SEGNALE CHIUSURA PORTA TAGLIAFUOCO
   E119 AT %M114.6 : Bool;   // [B2782] CONTROLLO 1 POSIZIONAMENTO POS. 05
   E120 AT %M114.7 : Bool;   // [B2783] CONTROLLO 2 POSIZIONAMENTO POS. 05
   E121 AT %M115.0 : Bool;   // Pallet ready in infeed signal (Infeed signal)
   E122 AT %M115.1 : Bool;   // Ready to receive pallet from outfeed signal (Outfeed signal)
   E123 AT %M115.2 : Bool;   // End of pallet transfer signal (Outfeed signal)
   E124 AT %M115.3 : Bool;
   In_Pos1 AT %M116.0 : Bool;   // Conveyor pos.1 positioning support memory
   In_Forklift1 AT %M116.1 : Bool;   // Forklift presence conveyor pos.1 (support memory)
   In_Pos2 AT %M116.4 : Bool;   // Conveyor pos.2 positioning support memory
   In_Pos3 AT %M117.0 : Bool;   // Conveyor pos.3 positioning support memory
   A01 AT %M120.0 : Bool;   // Request to open door (Technoplat)
   A02 AT %M120.1 : Bool;   // Rele' on pilz chain (Technoplat)
   A03 AT %M120.2 : Bool;   // Emergency mode lamp (Technoplat)
   A04 AT %M120.3 : Bool;   // Automatic mode lamp (Technoplat)
   A05 AT %M120.4 : Bool;   // Film ended or broken lamp (Technoplat)
   A06 AT %M120.5 : Bool;   // Acoustic signal (Technoplat)
   A07 AT %M120.6 : Bool;   // Forward on table rotation inverter (Technoplat)
   A08_NotUsed AT %M120.7 : Bool;   // Speed selection (X2-S4I) on arm rotation inverter (Technoplat)
   A09_NotUsed AT %M121.0 : Bool;   // Speed selection (X3-S5I) on arm rotation inverter (Technoplat)
   A10 AT %M121.1 : Bool;   // Backward on table rotation inverter (Technoplat)
   A11 AT %M121.2 : Bool;   // Motor and brake for table rotation motor (Technoplat)
   A12 AT %M121.3 : Bool;   // Brake for table rotation motor (Technoplat)
   A13 AT %M121.4 : Bool;   // Forward on spool carriage(upward) and machine conveyor inverter (Technoplat)
   A14 AT %M121.5 : Bool;   // Backward on spool carriage(downward) and machine conveyor inverter (Technoplat)
   A15 AT %M121.6 : Bool;   // Spool carriage prestretch motor (Prestretch)
   A16 AT %M121.7 : Bool;   // Positioning command for OFF3 U201 (ON=normal functioning/OFF fast stop)
   A17_NotUsed AT %M122.0 : Bool;   // Pallet lifter upward(1)/downard (Lifter)
   A18_NotUsed AT %M122.1 : Bool;   // Pressure plate upward/downward(1) (Pressure plate)
   A19 AT %M122.2 : Bool;   // Opening/closing(1) single rope unit (Rope unit)
   A20 AT %M122.3 : Bool;   // Motor for spool carriage (Technoplat)
   A21_NotUsed AT %M122.4 : Bool;   // Jog1 speed for fast prestretch rool (Prestretch)
   A22_NotUsed AT %M122.5 : Bool;   // EN1 for fast prestretch rool (Prestretch)
   A23 AT %M122.6 : Bool;   // Opening/closing(1) lower (double) rope unit (Rope unit)
   A24 AT %M122.7 : Bool;   // Pressure plate upward (Technoplat pressure plate)
   A25 AT %M123.0 : Bool;   // Pressure plate downward (Technoplat pressure plate)
   A26 AT %M123.1 : Bool;   // Opening/closing(2) lower(double) rope unit (Rope unit)
   A27_NotUsed AT %M123.2 : Bool;
   A28 AT %M123.3 : Bool;   // LedBypass
   A29 AT %M123.4 : Bool;   // Enable (EN) for arm rotation and top inverter
   A30 AT %M123.5 : Bool;   // Motor for machine conveyor (Technoplat)
   A31_NotUsed AT %M123.6 : Bool;
   A32 AT %M123.7 : Bool;   // Ready to receive pallet from infeed signal reverse cycle
   A33 AT %M124.0 : Bool;   // End of pallet transfer from infeed signal reverse cycle
   A34 AT %M124.1 : Bool;   // Ready to receive pallet from infeed signal (Std signal)
   A35 AT %M124.2 : Bool;   // End of pallet transfer from infeed signal (Std signal)
   A36 AT %M124.3 : Bool;   // Pallet ready for outfeed signal (Std signal)
   A37_NotUsed AT %M124.4 : Bool;   // Motor for infeed conveyor (Conveyor)
   A38 AT %M124.5 : Bool;   // Machine in position signal (No conveyor signal)
   A39 AT %M124.6 : Bool;   // Wrapp ended signal (No conveyor signal)
   A40_NotUsed AT %M124.7 : Bool;
   A41_NotUsed AT %M125.0 : Bool;   // Film clamp upward (RingSpring clamp)
   A42_NotUsed AT %M125.1 : Bool;   // Film clamp downward (RingSpring clamp)
   A43_NotUsed AT %M125.2 : Bool;   // Film clamp opening(1)/closing (RingSpring clamp)
   A44 AT %M125.3 : Bool;   // Welder contrast upward(1)/downward (RingSpring clamp)
   A45_NotUsed AT %M125.4 : Bool;   // Welder unit upward(1)/downward (RingSpring clamp)
   A46 AT %M125.5 : Bool;   // Film cutter wire on (All clamp)
   A47 AT %M125.6 : Bool;   // Film welder on (All clamp)
   A48_NotUsed AT %M125.7 : Bool;   // Welder unit cooler (RingSpring clamp)
   A49 AT %M126.0 : Bool;   // Airblower for film tail (All clamp)
   A50 AT %M126.1 : Bool;   // Cutting and welding unit forward(1)/backward (Claw clamp)
   A51 AT %M126.2 : Bool;   // Film clamp opening (Claw clamp)
   A52 AT %M126.3 : Bool;   // Film clamp closing (Claw clamp)
   A53_NotUsed AT %M126.4 : Bool;   // Film clamp double closing (Claw clamp)
   A54_NotUsed AT %M126.5 : Bool;   // Welder unit forward(1)/backward (Claw clamp)
   A55_NotUsed AT %M126.6 : Bool;   // Film clamp carriage forward (Spring clamp)
   A56_NotUsed AT %M126.7 : Bool;   // Film clamp carriage backward (Spring clamp)
   A57 AT %M127.0 : Bool;   // Welder contrast forward (Contrast carriage)
   A58 AT %M127.1 : Bool;   // Welder contrast backward (Contrast carriage)
   A59 AT %M127.2 : Bool;   // Table position to open clamp during wrapping cycle
   A60 AT %M127.3 : Bool;
   A61 AT %M127.4 : Bool;
   A62 AT %M127.5 : Bool;
   A63 AT %M127.6 : Bool;   // Infeed safety barrier muting for muting by plc (Barrier)
   A64 AT %M127.7 : Bool;   // Outfeed safety barrier muting for muting by plc (Barrier)
   A65 AT %M128.0 : Bool;   // Signal ready to receive pallet from infeed (Infeed signal)
   A66 AT %M128.1 : Bool;   // Signal end of pallet transfer from infeed (Infeed signal)
   A67 AT %M128.2 : Bool;   // Signal pallet ready for outfeed (Outfeed signal)
   A68 AT %M128.3 : Bool;   // SEGNALE PRONTO PER CHIUSURA PORTA TAGLIAFUOCO
   A69 AT %M128.4 : Bool;
   A70 AT %M128.5 : Bool;
   A71 AT %M128.6 : Bool;
   A72 AT %M128.7 : Bool;
   A73 AT %M129.0 : Bool;
   A74 AT %M129.1 : Bool;
   A75 AT %M129.2 : Bool;   // Top carriage upward (Top)
   A76 AT %M129.3 : Bool;   // Top carriage downward (Top)
   A77 AT %M129.4 : Bool;   // Top carriage forward (Top)
   A78 AT %M129.5 : Bool;   // Top carriage backward (Top)
   A79 AT %M129.6 : Bool;   // Top cutter forward (Top)
   A80 AT %M129.7 : Bool;   // Top cutter backward (Top)
   A81 AT %M130.0 : Bool;   // Closing clamp to block top film (Top)
   A82 AT %M130.1 : Bool;   // Opening clamp to block top film (Top)
   A83 AT %M130.2 : Bool;   // Closing clamp to lift(pull) top film (Top)
   A84 AT %M130.3 : Bool;   // Opening clamp to lift(pull) top film (Top)
   A85 AT %M130.4 : Bool;   // Top carriage brake (Top)
   A86 AT %M130.5 : Bool;
   A87 AT %M130.6 : Bool;
   A88 AT %M130.7 : Bool;
   Clock01 AT %M255.0 : Bool;   // Clock 0,1 seconds (Period)
   Clock02 AT %M255.1 : Bool;   // Clock 0,2 seconds (Period)
   Clock04 AT %M255.2 : Bool;   // Clock 0,4 seconds (Period)
   Clock05 AT %M255.3 : Bool;   // Clock 0,5 seconds (Period)
   Clock08 AT %M255.4 : Bool;   // Clock 0,8 seconds (Period)
   Clock10 AT %M255.5 : Bool;   // Clock 1,0 seconds (Period)
   Clock16 AT %M255.6 : Bool;   // Clock 1,6 seconds (Period)
   Clock20 AT %M255.7 : Bool;   // Clock 2,0 seconds (Period)
   MB0 AT %MB0 : Byte;   // Machine cycle (1) byte
   MB1 AT %MB1 : Byte;   // Machine cycle (2) byte
   MW2 AT %MW2 : Word;   // Machine cycle (3) word
   MB5 AT %MB5 : Byte;   // Top cycle (1) byte
   MW6 AT %MW6 : Word;   // Top cycle (2) word
   MW8 AT %MW8 : Word;   // Top film ended cycle word
   Tag_9 AT %M8.7 : Bool;
   MB16 AT %MB16 : Byte;   // Conveyor cycle byte
   MB17 AT %MB17 : Byte;   // Pallet load cycle byte
   MB20 AT %MB20 : Byte;   // Claw clamp HS40 cycle byte
   MB24 AT %MB24 : Byte;
   MB30 AT %MB30 : Byte;   // Film broken cycle byte
   MB32 AT %MB32 : Byte;   // Film broken cycle 1 byte
   In_Forklift2 AT %M116.5 : Bool;   // Forklift presence conveyor pos.2 (support memory)
   V50_0 AT %M50.0 : Bool;   // Support for end of transfer signal
   V50_2 AT %M50.2 : Bool;   // Transit memory pos1->pos2
   V51_2 AT %M51.2 : Bool;   // Memory to exclude wrapping in pos 2
   In_Pos4 AT %M117.4 : Bool;   // Conveyor pos.4 positioning support memory
   In_Forklift4 AT %M117.5 : Bool;   // Forklift presence conveyor pos.4 (support memory)
   V52_0 AT %M52.0 : Bool;   // Transit memory pos3->pos4
   V50_4 AT %M50.4 : Bool;   // Transit memory pos3->pos4
   V52_1 AT %M52.1 : Bool;   // Outfeed conveyor pos.4 unload
   V50_5 AT %M50.5 : Bool;   // Transit memory pos4->pos5
   "M1.4_N" AT %M200.0 : Bool;   // Negative edge M1.4
   V50_3 AT %M50.3 : Bool;   // Transit memory pos2->pos3
   In_Forklift3 AT %M117.1 : Bool;   // Forklift presence conveyor pos.3 (support memory)
   Off AT %M12.6 : Bool;   // Bit always off
   U201_Start AT %M161.0 : Bool;
   U201_Ack AT %M161.1 : Bool;
   U201_Rev AT %M161.2 : Bool;
   U221_Start AT %M161.3 : Bool;
   U221_Ack AT %M161.4 : Bool;
   U221_Rev AT %M161.5 : Bool;
   U241_Start AT %M161.6 : Bool;
   U241_Ack AT %M161.7 : Bool;
   U241_Rev AT %M162.0 : Bool;
   U261_Start AT %M162.1 : Bool;
   U261_Ack AT %M162.2 : Bool;
   U261_Rev AT %M162.3 : Bool;
   U321_Start AT %M162.4 : Bool;
   U321_Ack AT %M162.5 : Bool;
   U321_Rev AT %M162.6 : Bool;
   U201_OFF1 AT %M170.0 : Bool;
   U201_OFF3 AT %M170.1 : Bool;
   U321_OFF1 AT %M170.2 : Bool;
   U321_OFF3 AT %M170.3 : Bool;
   InverterFail AT %M163.0 : Bool;   // Inverter Fault/Alarm - Anomalia/Avviso
   InverterFault AT %M163.1 : Bool;   // Inverter Fault (F) - Anomalia
   InverterAlarm AT %M163.2 : Bool;   // Inverter Alarm (A) - Avviso
   PrestNewValue AT %M160.0 : Bool;
   System_Byte AT %MB254 : Byte;
   FirstScan AT %M254.0 : Bool;
   DiagStatusUpdate AT %M254.1 : Bool;
   AlwaysTRUE AT %M254.2 : Bool;
   AlwaysFALSE AT %M254.3 : Bool;
   U201_Start_ARM AT %M170.6 : Bool;
   U201_Start_RUL AT %M170.7 : Bool;
   U201_Feedback AT %M171.0 : Bool;   // Feedback motori sotto inverter U201 (braccio/rull.CM)
   U221_Feedback AT %M171.1 : Bool;   // Feedback motore sotto inverter U221 (carrello)
   U241_Feedback AT %M171.2 : Bool;   // Feedback motore sotto inverter U241 (tiro)
   U261_Feedback AT %M171.3 : Bool;   // Feedback motore sotto inverter U261 (prestiro)
   Tag_14 AT %M13.2 : Bool;
   Tag_10 AT %M14.5 : Bool;
   CELLA AT %MW145 : Int;   // Valore cella di carico (modbus)
   ResetLoadCell AT %M144.7 : Bool;   // "DB100_Display".ResetLoadCell
   ERR AT %MD155 : DInt;   // Errore (SP-feedback)
   PROVA AT %MD150 : DWord;
   BitClock1 AT %M143.1 : Bool;   // Impulso ogni 20ms (OB30)
   BitClock2 AT %M143.2 : Bool;   // Impulso ogni 100ms (OB30 x5)
   In_Pos5 AT %M117.6 : Bool;   // Conveyor pos.5 positioning support memory
   In_Pos6 AT %M117.7 : Bool;   // Conveyor pos.6 positioning support memory
   In_Pos7 AT %M118.0 : Bool;   // Conveyor pos.7 positioning support memory
   In_Pos8 AT %M118.1 : Bool;   // Conveyor pos.8 positioning support memory
   V50_7 AT %M50.7 : Bool;   // Transit memory pos7->pos8
   V51_0 AT %M51.0 : Bool;   // Outfeed conveyor pos.8 unload
   V51_3 AT %M51.3 : Bool;   // Memory to exclude wrapping in pos 3
   V51_4 AT %M51.4 : Bool;   // Memory to exclude wrapping in pos 4
   V51_5 AT %M51.5 : Bool;   // Memory to exclude wrapping in pos 5
END_VAR
